{attribute 'conditionalshow'}
TYPE INTERNAL ST_ScopedContextStack :
STRUCT
	aScopedContext		: ARRAY[0..Config.nMaxScopedContext-1] OF I_ContextBuilder;
	nScopeContextCount	: UINT (0..Config.nMaxScopedContext);
END_STRUCT
END_TYPE

(* stored: Version 1.1.0.1, ProductVersion 3.1.4024.6
   DUT ST_ScopedContextStack: Id {4a8187ff-c55a-454e-89ac-86e2dc158433} *)
